FUNCTION_BLOCK Motorsteuerung
VAR_INPUT
END_VAR
VAR_OUTPUT
END_VAR
VAR
END_VAR

// NETWORK 1

END_FUNCTION_BLOCK

(* stored: Version 1.1.0.1, ProductVersion 3.1.4022.3
   POU Motorsteuerung: Id {04423fcb-67e2-4151-aa33-55f5a4a69b98}, SpecialFunc None *)
